// TIA Portal V19 export
TYPE "LEXCHANGETRAY_typeRollerVfdInterface"
// commandConfiguration: LEXCHANGETRAY_typeRollerVfdContronNodeCommandConfiguration
// commands: LEXCHANGETRAY_typeRollerVfdManualCommands
// monitoring: LEXCHANGETRAY_typeVfdProcessValues
// configuration: LBC_typeSinaSpeedConfiguration
// stored: Access Published
   STRUCT
      commandConfiguration : "LEXCHANGETRAY_typeRollerVfdContronNodeCommandConfiguration";
      commands { S7_SetPoint := 'True'} : "LEXCHANGETRAY_typeRollerVfdManualCommands";
      monitoring { S7_SetPoint := 'True'} : "LEXCHANGETRAY_typeVfdProcessValues";
      configuration : "LBC_typeSinaSpeedConfiguration";
   END_STRUCT;
END_TYPE
